(* PLC project piece, Dassault Systèmes ControlBuild 2024x *)
(* stored: creationDateTime 2023-10-03T11:13:43-01:00 *)

FUNCTION_BLOCK drill.piece
  VAR_INPUT
    loadingRequest : BOOL := false;
    unloadingRequest : BOOL := false;
  END_VAR
  VAR_OUTPUT
    piece : BOOL := false;
  END_VAR
  VAR
    count : DINT := 0;
  END_VAR
  VAR CONSTANT
    loadingDuration : DINT := 10;
  END_VAR


ACTION C_source_code:
if (loadingRequest)
   {
   piece = 1;
   count = 0;
   }
if (unloadingRequest)
   {
   count = count+1;
   if (count == loadingDuration) piece=0;
   }
END_ACTION
END_FUNCTION_BLOCK
